PROGRAM MAIN_UDP
VAR
	//sPaketinhalt	: LREAL;
	//nPaketlaenge	: UDINT;
	
	x	  AT%Q*	: ARRAY[1..4] OF LREAL;
	y	  AT%Q*	: ARRAY[1..4] OF LREAL;
	theta AT%Q*	: ARRAY[1..4] OF LREAL;
	udp1 : UDPConnect;
END_VAR

udp1();

END_PROGRAM

(* stored: Version 1.1.0.1, ProductVersion 3.1.4022.3
   POU MAIN_UDP: Id {b6e4ea55-b300-41b8-8a89-a1df4d8038ad}, SpecialFunc None *)
